FUNCTION_BLOCK FB_BlockPad
VAR_INPUT
	iInput1 : BOOL;
	iInput2 : BOOL;
	iInput3 : BOOL;
END_VAR
VAR_OUTPUT
	
	Q : BOOL;
	oLight1 : BOOL;
	
END_VAR
VAR
END_VAR


iInput1;
iInput2;
oLight1;

END_FUNCTION_BLOCK

(* stored: Version 1.1.0.1, ProductVersion 3.1.4024.10
   POU FB_BlockPad: Id {718ab21c-a86f-42b1-ad84-7eea86241524}, SpecialFunc None *)
